FUNCTION MotorAngularVelocityToCableVelocity : LREAL
VAR_INPUT
	motor_velocity : LREAL;
END_VAR
VAR_OUTPUT
	cable_velocity : LREAL;
END_VAR
VAR
END_VAR

cable_velocity := motor_velocity;

END_FUNCTION

(* stored: Version 1.1.0.1, ProductVersion 3.1.4024.11
   POU MotorAngularVelocityToCableVelocity: Id {c1aa46c1-63df-4cf7-884e-dbfb053fb6ea}, SpecialFunc None *)
